{attribute addProperty BoxType "EL3102-0000-0019"}
{attribute addProperty Id "StatusAT %I*Status_84521898587.251ValueAT %I*INT16217"}
{attribute addProperty CRC "1839201807"}
{attribute addProperty SizeInBites "74"}
{attribute addProperty SizeInBytes "9.25"}
TYPE AI_Standard_Channel_6D9FFE0F :
STRUCT
	{attribute addProperty Name "Status"}
	Status AT %I* : Status_84521898;
	{attribute addProperty Name "Value"}
	Value AT %I* : INT;
END_STRUCT
END_TYPE

(* stored: Version 1.2.0.0, ProductVersion 3.1.4024.9
   DUT AI_Standard_Channel_6D9FFE0F: Id {c356ffa3-9f1e-4baf-a2a2-2bd31c460ee2} *)
